{attribute 'strict'}
TYPE E_CognexCameraGetValueSpreadsheetStatus :
(
	WAITING_FOR_STATUS_CODE						:= 2,
	THE_COMMAND_WAS_EXECUTED_SUCCESSFULLY		:= 1,
	UNRECOGNIZED_COMMAND 						:= 0,
	THE_CELL_ID_IS_INVALID						:= -1,
	THE_COMMAND_COULD_NOT_BE_EXECUTED 			:= -2
);
END_TYPE

(* stored: Version 1.1.0.1, ProductVersion 3.1.4024.9
   DUT E_CognexCameraGetValueSpreadsheetStatus: Id {41ce4f7b-651e-4468-b452-667497dc7274} *)
